RoboDK station: picknplace using palletizing.rdk

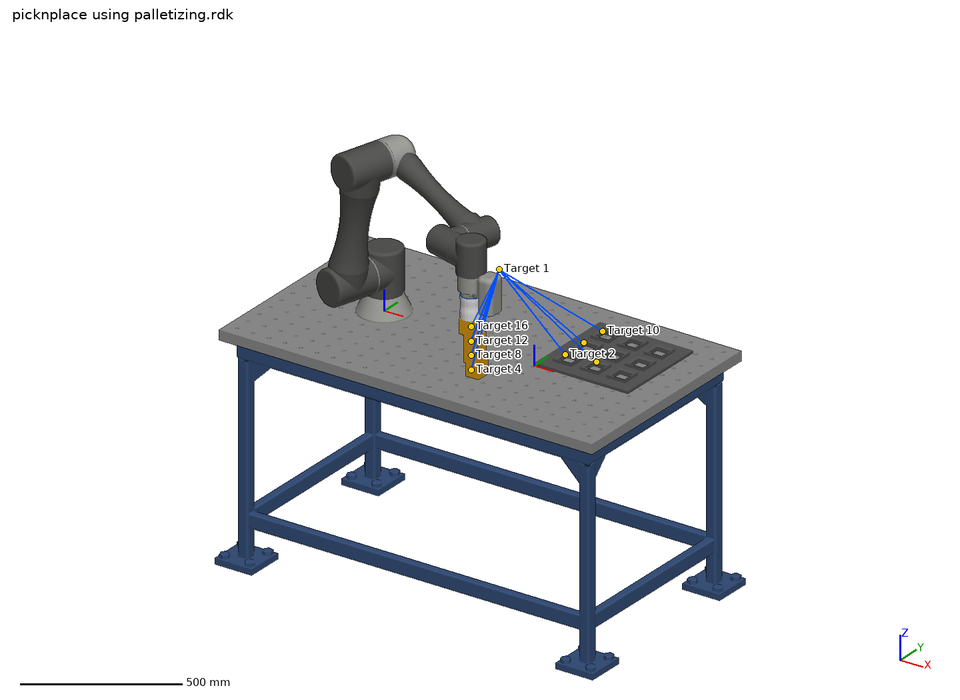
[picture v0: the station drawn from its stored meshes, robots at their saved joint values, targets as dots, program paths as lines]
Station picknplace using palletizing (saved by RoboDK 5.7.5). Poses are relative to the parent item; angles as X-Y-Z fixed-axis rotations.
  - frame TM5-900 Base at (0, 0, 0) mm
    - robot TM5-900: 6 axes, payload 4 kg, reach 900 mm, repeatability 0.1 mm, weight 30 kg
        modified DH rows (alpha deg, a mm, theta deg, d mm): 0, 0, 0, 145.2; 90, 0, 90, 0; 0, 429, 0, 0; 0, 411, -90, 122.3; -90, 0, 0, 106.5; 90, 0, 180, 114.15
        joint limits [-360, -180, -155, -180, -180, -270] to [360, 180, 155, 180, 180, 270]; home [0, 0, 90, -90, 90, 0]; saved at [-15.68, 10.058, 98.154, -18.213, 90, -15.68]
      - tool OnRobot MG10 Magnetic Gripper, TCP at (0, 0, 93) mm, size 71 x 74.9 x 91.4 mm
  - object Table 1400x800x800mm at (0, 0, 0) mm, size 1420 x 820 x 800 mm, geometry from Table-1400x800x800mm.sld
  - frame Frame 2 at (600, -50, 0) mm
    - target Target 1 (Cartesian target) at (-82.5, -72.3, 335.05) mm, rotated rx 180 ry 0 rz 90 deg; joints [0, 0, 90, 0, 90, 0] of TM5-900
    - object Pallete  at (0, 0, 0) mm, size 350 x 350 x 20 mm, geometry from Pallete .step
    - target Target 2 (Cartesian target) at (67.5, 67.7, 30.05) mm, rotated rx 180 ry 0 rz 90 deg; joints [12.073, 30.79, 95.721, -36.511, 90, 12.073] of TM5-900
    - target Target 3 (Cartesian target) at (-82.5, -72.3, 335.05) mm, rotated rx 180 ry 0 rz 90 deg; joints [0, 0, 90, 0, 90, 0] of TM5-900
    - target Target 4 (Cartesian target) at (-82.5, -222.3, 50) mm, rotated rx 180 ry 0 rz 90 deg; joints [-15.68, 19.959, 109.154, -39.113, 90, -15.68] of TM5-900
    - target Target 5 (Cartesian target) at (-82.5, -72.3, 335.05) mm, rotated rx 180 ry 0 rz 90 deg; joints [0, 0, 90, 0, 90, 0] of TM5-900
    - target Target 6 (Cartesian target) at (67.5, 167.7, 30.05) mm, rotated rx 180 ry 0 rz 90 deg; joints [20.395, 31.897, 93.869, -35.766, 90, 20.395] of TM5-900
    - target Target 7 (Cartesian target) at (-82.5, -72.3, 335.05) mm, rotated rx 180 ry 0 rz 90 deg; joints [0, 0, 90, 0, 90, 0] of TM5-900
    - target Target 8 (Cartesian target) at (-82.5, -222.3, 100) mm, rotated rx 180 ry 0 rz 90 deg; joints [-15.68, 15.875, 106.272, -32.147, 90, -15.68] of TM5-900
    - target Target 9 (Cartesian target) at (-82.5, -72.3, 335.05) mm, rotated rx 180 ry 0 rz 90 deg; joints [0, 0, 90, 0, 90, 0] of TM5-900
    - target Target 10 (Cartesian target) at (67.5, 267.7, 30.05) mm, rotated rx 180 ry 0 rz 90 deg; joints [28.095, 34.606, 89.271, -33.877, 90, 28.095] of TM5-900
    - target Target 11 (Cartesian target) at (-82.5, -72.3, 335.05) mm, rotated rx 180 ry 0 rz 90 deg; joints [0, 0, 90, 0, 90, 0] of TM5-900
    - target Target 12 (Cartesian target) at (-82.5, -222.3, 150) mm, rotated rx 180 ry 0 rz 90 deg; joints [-15.68, 12.568, 102.598, -25.165, 90, -15.68] of TM5-900
    - target Target 13 (Cartesian target) at (-82.5, -72.3, 335.05) mm, rotated rx 180 ry 0 rz 90 deg; joints [0, 0, 90, 0, 90, 0] of TM5-900
    - target Target 14 (Cartesian target) at (177.5, 77.7, 30.05) mm, rotated rx 180 ry 0 rz 90 deg; joints [11.085, 43.576, 73.455, -27.031, 90, 11.085] of TM5-900
    - target Target 15 (Cartesian target) at (-82.5, -72.3, 335.05) mm, rotated rx 180 ry 0 rz 90 deg; joints [0, 0, 90, 0, 90, 0] of TM5-900
    - target Target 16 (Cartesian target) at (-82.5, -222.3, 200) mm, rotated rx 180 ry 0 rz 90 deg; joints [-15.68, 10.058, 98.154, -18.213, 90, -15.68] of TM5-900
    - target Target 17 (Cartesian target) at (-82.5, -72.3, 335.05) mm, rotated rx 180 ry 0 rz 90 deg; joints [0, 0, 90, 0, 90, 0] of TM5-900
  - program Prog1 (26 instructions, listed below)
  - program Prog2 (3 instructions, listed below)
  - object Cube 50mm at (500, -280, 29.95) mm, size 50 x 50 x 50 mm, geometry from Cube-50mm.sld
  - object Cube 50mm at (500, -290, 79.95) mm, size 50 x 50 x 50 mm, geometry from Cube-50mm (3).sld
  - object Cube 50mm at (500, -290, 129.95) mm, size 50 x 50 x 50 mm, geometry from Cube-50mm (3).sld
  - object Cube 50mm at (490, -300, 179.95) mm, size 50 x 50 x 50 mm, geometry from Cube-50mm (3).sld
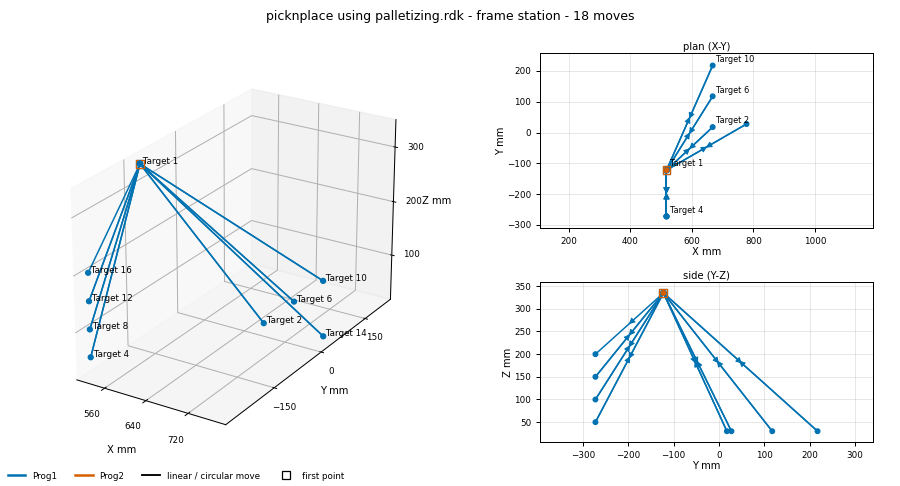
[picture p0: tool path of picknplace using palletizing.rdk in frame station, 18 of 18 moves have a stored position in this frame; points joined in program order, loops and branches not executed]

--- program Prog1 (robot TM5-900) ---
  Set Ref.: Frame 2
  MoveJ (Target 1)
  MoveL (Target 1)
  MoveL (Target 2)
  Attach to OnRobot MG10 Magnetic Gripper
  MoveL (Target 3)
  MoveL (Target 4)
  Detach from OnRobot MG10 Magnetic Gripper
  MoveL (Target 5)
  MoveL (Target 6)
  Attach to OnRobot MG10 Magnetic Gripper
  MoveL (Target 7)
  MoveL (Target 8)
  Detach from OnRobot MG10 Magnetic Gripper
  MoveL (Target 9)
  MoveL (Target 10)
  Attach to OnRobot MG10 Magnetic Gripper
  MoveL (Target 11)
  MoveL (Target 12)
  Detach from OnRobot MG10 Magnetic Gripper
  MoveL (Target 13)
  MoveL (Target 14)
  Attach to OnRobot MG10 Magnetic Gripper
  MoveL (Target 15)
  MoveL (Target 16)
  Detach from OnRobot MG10 Magnetic Gripper

--- program Prog2 (robot TM5-900) ---
  Set Ref.: Frame 2
  MoveL (Target 17)
  Replace objects
